(* CODESYS project EX3.project

Project tree, tasks and I/O mapping:
  Device : CODESYS Control Win V3, 3S - Smart Software Solutions GmbH, order no. 305021, version 3.5.11.30
    application Application
      libraries: Standard, * (System)
      task MainTask (cyclic, interval t#20ms, priority 1) calls PLC_PRG
      program PLC_PRG [LD]
*)

// Device/Application/PLC_PRG
PROGRAM PLC_PRG
VAR
	BT1 : BOOL;       // LIGA SISTEMA
	BT2 : BOOL;       // DESLIGA SISTEMA
	LAMP1 : BOOL;     // INDICA FUNCIONAMENTO DO SISTEMA
	TON_1: TON;       // VARIAVEL TIPO TON TON 1
	ET0: TIME;        // VARIAVEL TIPO TIME TON 1
	KM1: BOOL;        // TRIANGULO
	KT1: BOOL;        // SENSOR DE PROTECAO
	KM2: BOOL;        // ESTELA
	KM3: BOOL;
	TON_2: TON;      // VARIAVEL TIPO TON TON 2
	ET1: TIME;       // VARIAVEL TIPO TIME TON 2
END_VAR

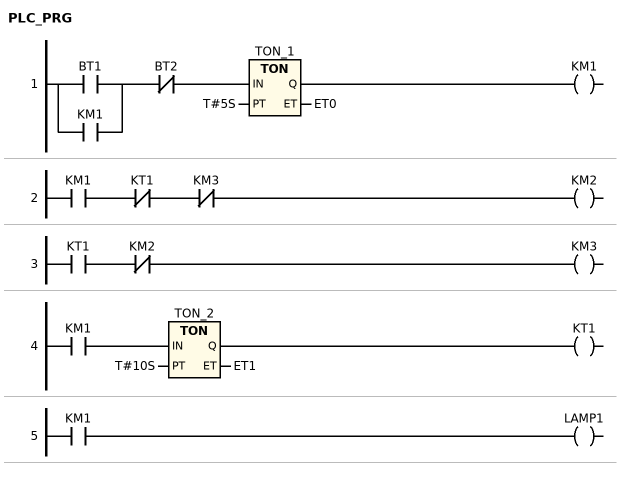
// NETWORK 1
TON_1(IN := (BT1 OR KM1) AND NOT BT2, PT := T#5S, ET => ET0); // TON
KM1 := TON_1.Q;

// NETWORK 2
KM2 := KM1 AND NOT KT1 AND NOT KM3;

// NETWORK 3
KM3 := KT1 AND NOT KM2;

// NETWORK 4
TON_2(IN := KM1, PT := T#10S, ET => ET1); // TON
KT1 := TON_2.Q;

// NETWORK 5
LAMP1 := KM1;

END_PROGRAM
